TYPE ST_KeyenceLaser_TwoD_Code_Read_Result :
STRUCT
Marking_Check_Score_TwoDC_Read_Grade_Status		: WORD ;
Check_Count_Status								: WORD ;
ReserveDWord_2									: DWORD ;
END_STRUCT
END_TYPE

(* stored: Version 1.1.0.1, ProductVersion 3.1.4024.11
   DUT ST_KeyenceLaser_TwoD_Code_Read_Result: Id {c759ce13-2577-4a13-8369-bba07e7ccdeb} *)
